// TIA Portal V17 export
// export: Created 2025-06-26T07:49:36.6585536Z, ExportSetting WithDefaults, DisplayName Totally Integrated Automation Portal, DisplayVersion V17 Update 8, DisplayName TIA Portal Openness, DisplayVersion V17 Update 8, DisplayName TIA Portal Version Control Interface, DisplayVersion V17, DisplayName STEP 7 Professional, DisplayVersion V17 Update 8, DisplayName STEP 7 Safety, DisplayVersion V17 Update 6, DisplayName WinCC Advanced, DisplayVersion V17 Update 8
FUNCTION_BLOCK "InputWarningHandling"   // FB7, FBD
TITLE = Handle I/O warnings
{ S7_Optimized_Access := 'TRUE' }
AUTHOR : Heaten
VERSION : 0.1
// stored: AutoNumber false, IsIECCheckEnabled false, IsRetainMemResEnabled false, MemoryReserve 100, SetENOAutomatically false, UDAEnableTagReadback false
   VAR
      A1101 { ExternalAccessible := 'False'; ExternalVisible := 'False'; ExternalWritable := 'False'; S7_SetPoint := 'True'} : "fbDigitalAlarm";
      A1121 { ExternalAccessible := 'False'; ExternalVisible := 'False'; ExternalWritable := 'False'; S7_SetPoint := 'True'} : "fbDigitalAlarm";
      A1140 { ExternalAccessible := 'False'; ExternalVisible := 'False'; ExternalWritable := 'False'; S7_SetPoint := 'True'} : "fbDigitalAlarm";
      A1216 { ExternalAccessible := 'False'; ExternalVisible := 'False'; ExternalWritable := 'False'; S7_SetPoint := 'True'} : "fbHMIEvent";
      A1217 { ExternalAccessible := 'False'; ExternalVisible := 'False'; ExternalWritable := 'False'; S7_SetPoint := 'True'} : "fbHMIEvent";
      A1218 { ExternalAccessible := 'False'; ExternalVisible := 'False'; ExternalWritable := 'False'; S7_SetPoint := 'True'} : "fbHMIEvent";
      A1224 { ExternalAccessible := 'False'; ExternalVisible := 'False'; ExternalWritable := 'False'; S7_SetPoint := 'True'} : "fbHMIEvent";
      A1225 { ExternalAccessible := 'False'; ExternalVisible := 'False'; ExternalWritable := 'False'; S7_SetPoint := 'True'} : "fbHMIEvent";
      A1226 { ExternalAccessible := 'False'; ExternalVisible := 'False'; ExternalWritable := 'False'; S7_SetPoint := 'True'} : "fbHMIEvent";
      A1227 { ExternalAccessible := 'False'; ExternalVisible := 'False'; ExternalWritable := 'False'; S7_SetPoint := 'True'} : "fbHMIEvent";
      A1228 { ExternalAccessible := 'False'; ExternalVisible := 'False'; ExternalWritable := 'False'; S7_SetPoint := 'True'} : "fbHMIEvent";
      A1229 { ExternalAccessible := 'False'; ExternalVisible := 'False'; ExternalWritable := 'False'; S7_SetPoint := 'True'} : "fbHMIEvent";
      A1230 { ExternalAccessible := 'False'; ExternalVisible := 'False'; ExternalWritable := 'False'; S7_SetPoint := 'True'} : "fbHMIEvent";
      A1234 { ExternalAccessible := 'False'; ExternalVisible := 'False'; ExternalWritable := 'False'; S7_SetPoint := 'True'} : "fbHMIEvent";
      A1235 { ExternalAccessible := 'False'; ExternalVisible := 'False'; ExternalWritable := 'False'; S7_SetPoint := 'True'} : "fbHMIEvent";
      A1236 { ExternalAccessible := 'False'; ExternalVisible := 'False'; ExternalWritable := 'False'; S7_SetPoint := 'True'} : "fbHMIEvent";
      A1237 { ExternalAccessible := 'False'; ExternalVisible := 'False'; ExternalWritable := 'False'; S7_SetPoint := 'True'} : "fbHMIEvent";
      A1238 { ExternalAccessible := 'False'; ExternalVisible := 'False'; ExternalWritable := 'False'; S7_SetPoint := 'True'} : "fbHMIEvent";
      A1239 { ExternalAccessible := 'False'; ExternalVisible := 'False'; ExternalWritable := 'False'; S7_SetPoint := 'True'} : "fbHMIEvent";
      A1240 { ExternalAccessible := 'False'; ExternalVisible := 'False'; ExternalWritable := 'False'; S7_SetPoint := 'True'} : "fbHMIEvent";
      A1245 { ExternalAccessible := 'False'; ExternalVisible := 'False'; ExternalWritable := 'False'; S7_SetPoint := 'True'} : "fbHMIEvent";
      A1246 { ExternalAccessible := 'False'; ExternalVisible := 'False'; ExternalWritable := 'False'; S7_SetPoint := 'True'} : "fbHMIEvent";
      A1247 { ExternalAccessible := 'False'; ExternalVisible := 'False'; ExternalWritable := 'False'; S7_SetPoint := 'True'} : "fbHMIEvent";
      A1248 { ExternalAccessible := 'False'; ExternalVisible := 'False'; ExternalWritable := 'False'; S7_SetPoint := 'True'} : "fbHMIEvent";
      A1249 { ExternalAccessible := 'False'; ExternalVisible := 'False'; ExternalWritable := 'False'; S7_SetPoint := 'True'} : "fbHMIEvent";
      A1251 { ExternalAccessible := 'False'; ExternalVisible := 'False'; ExternalWritable := 'False'; S7_SetPoint := 'True'} : "fbHMIEvent";
      A1252 { ExternalAccessible := 'False'; ExternalVisible := 'False'; ExternalWritable := 'False'; S7_SetPoint := 'True'} : "fbHMIEvent";
      A1253 { ExternalAccessible := 'False'; ExternalVisible := 'False'; ExternalWritable := 'False'; S7_SetPoint := 'True'} : "fbHMIEvent";
      A1254 { ExternalAccessible := 'False'; ExternalVisible := 'False'; ExternalWritable := 'False'; S7_SetPoint := 'True'} : "fbHMIEvent";
      A1258 { ExternalAccessible := 'False'; ExternalVisible := 'False'; ExternalWritable := 'False'; S7_SetPoint := 'True'} : "fbHMIEvent";
      A1259 { ExternalAccessible := 'False'; ExternalVisible := 'False'; ExternalWritable := 'False'; S7_SetPoint := 'True'} : "fbHMIEvent";
      A1260 { ExternalAccessible := 'False'; ExternalVisible := 'False'; ExternalWritable := 'False'; S7_SetPoint := 'True'} : "fbHMIEvent";
      A1262 { ExternalAccessible := 'False'; ExternalVisible := 'False'; ExternalWritable := 'False'; S7_SetPoint := 'True'} : "fbHMIEvent";
      A1263 { ExternalAccessible := 'False'; ExternalVisible := 'False'; ExternalWritable := 'False'; S7_SetPoint := 'True'} : "fbHMIEvent";
      A1265 { ExternalAccessible := 'False'; ExternalVisible := 'False'; ExternalWritable := 'False'; S7_SetPoint := 'True'} : "fbHMIEvent";
      A1269 { ExternalAccessible := 'False'; ExternalVisible := 'False'; ExternalWritable := 'False'; S7_SetPoint := 'True'} : "fbHMIEvent";
      A1270 { ExternalAccessible := 'False'; ExternalVisible := 'False'; ExternalWritable := 'False'; S7_SetPoint := 'True'} : "fbHMIEvent";
      A1271 { ExternalAccessible := 'False'; ExternalVisible := 'False'; ExternalWritable := 'False'; S7_SetPoint := 'True'} : "fbHMIEvent";
      A1272 { ExternalAccessible := 'False'; ExternalVisible := 'False'; ExternalWritable := 'False'; S7_SetPoint := 'True'} : "fbHMIEvent";
      A1273 { ExternalAccessible := 'False'; ExternalVisible := 'False'; ExternalWritable := 'False'; S7_SetPoint := 'True'} : "fbHMIEvent";
      A1275 { ExternalAccessible := 'False'; ExternalVisible := 'False'; ExternalWritable := 'False'; S7_SetPoint := 'True'} : "fbHMIEvent";
      A1293 { ExternalAccessible := 'False'; ExternalVisible := 'False'; ExternalWritable := 'False'; S7_SetPoint := 'True'} : "fbHMIEvent";
      A1294 { S7_SetPoint := 'True'} : "fbDigitalAlarm";
      A1295 { S7_SetPoint := 'True'} : "fbDigitalAlarm";
      A3401 { ExternalAccessible := 'False'; ExternalVisible := 'False'; ExternalWritable := 'False'; S7_SetPoint := 'True'} : "fbDigitalAlarm";
      A5200 { ExternalAccessible := 'False'; ExternalVisible := 'False'; ExternalWritable := 'False'; S7_SetPoint := 'True'} : "fbHMIEvent";
      A5201 { ExternalAccessible := 'False'; ExternalVisible := 'False'; ExternalWritable := 'False'; S7_SetPoint := 'True'} : "fbHMIEvent";
      A5202 { ExternalAccessible := 'False'; ExternalVisible := 'False'; ExternalWritable := 'False'; S7_SetPoint := 'True'} : "fbHMIEvent";
      A5203 { ExternalAccessible := 'False'; ExternalVisible := 'False'; ExternalWritable := 'False'; S7_SetPoint := 'True'} : "fbDigitalAlarm";
      A5204 { ExternalAccessible := 'False'; ExternalVisible := 'False'; ExternalWritable := 'False'; S7_SetPoint := 'True'} : "fbDigitalAlarm";
      A5206 { ExternalAccessible := 'False'; ExternalVisible := 'False'; ExternalWritable := 'False'; S7_SetPoint := 'True'} : "fbHMIEvent";
      A5256 { ExternalAccessible := 'False'; ExternalVisible := 'False'; ExternalWritable := 'False'; S7_SetPoint := 'True'} : "fbHMIEvent";
   END_VAR
BEGIN

REGION Network 1: 1101
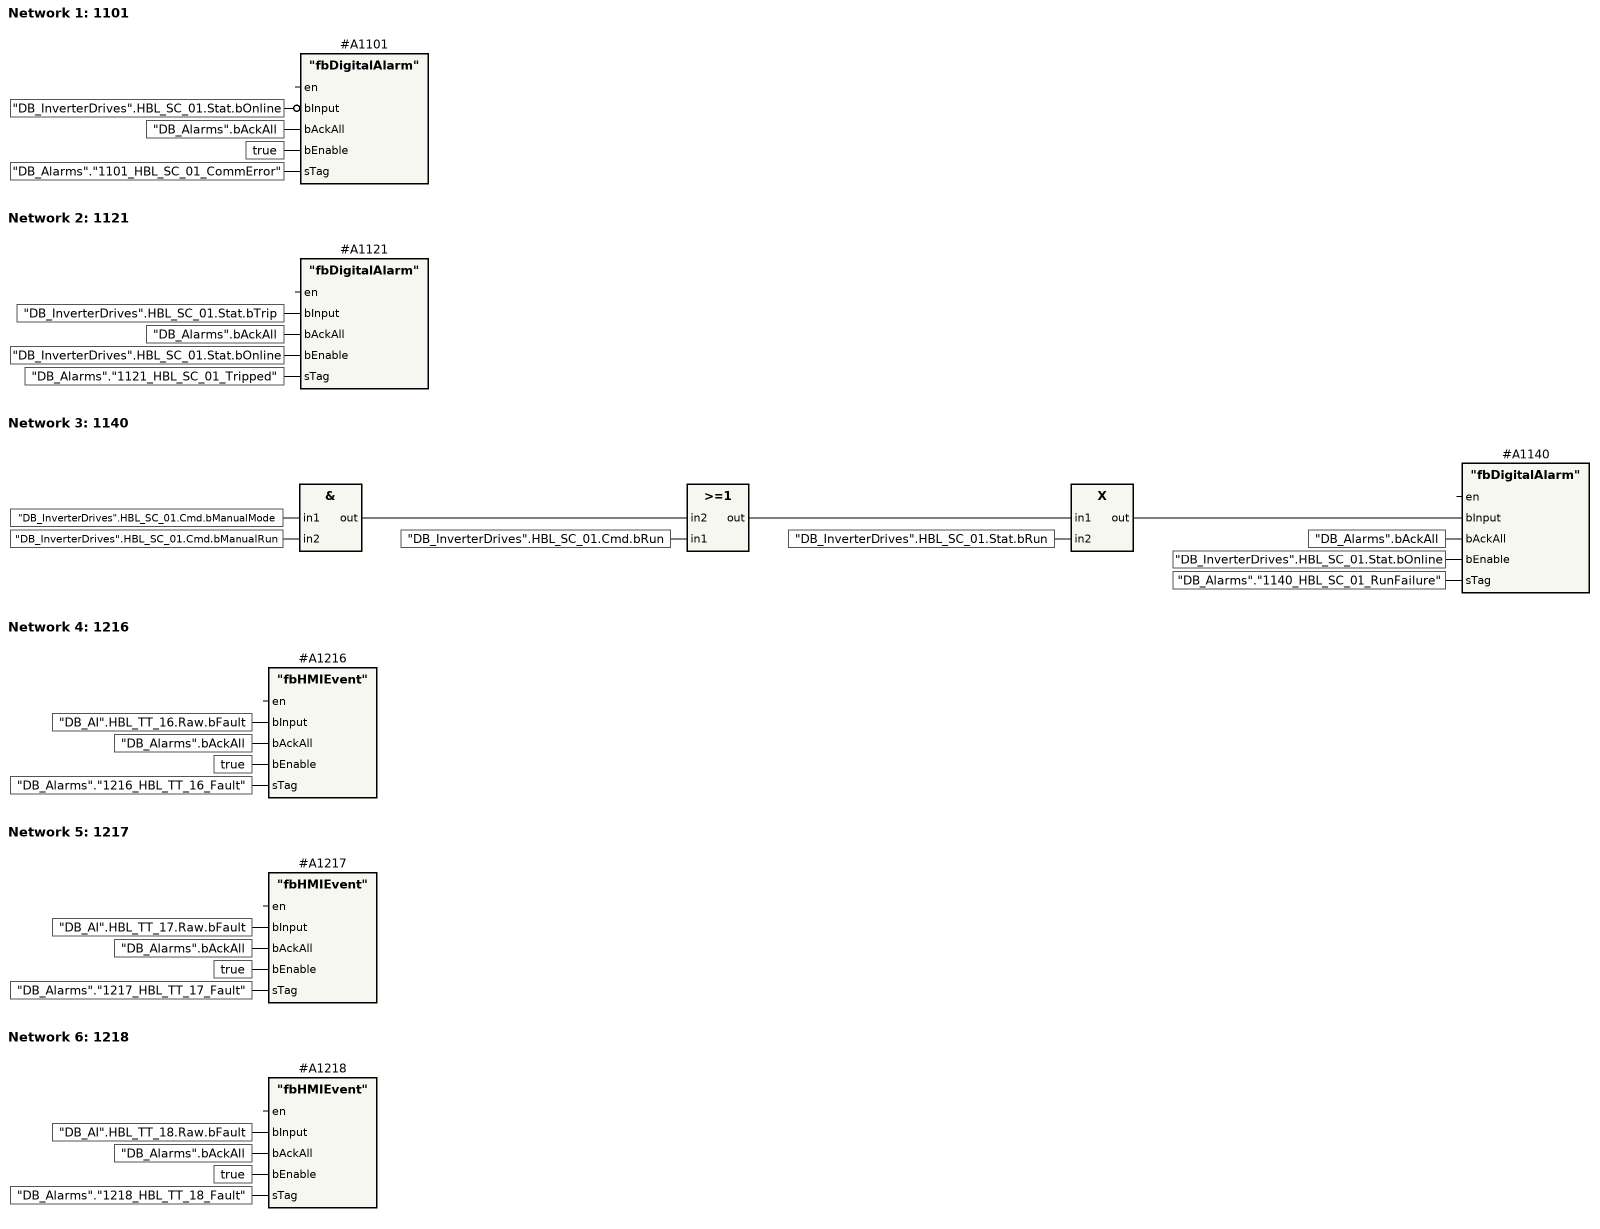
   #A1101(bInput := NOT "DB_InverterDrives".HBL_SC_01.Stat.bOnline,   // "fbDigitalAlarm"
          bAckAll := "DB_Alarms".bAckAll,
          bEnable := true,
          sTag := "DB_Alarms"."1101_HBL_SC_01_CommError");
END_REGION

REGION Network 2: 1121
   #A1121(bInput := "DB_InverterDrives".HBL_SC_01.Stat.bTrip,   // "fbDigitalAlarm"
          bAckAll := "DB_Alarms".bAckAll,
          bEnable := "DB_InverterDrives".HBL_SC_01.Stat.bOnline,
          sTag := "DB_Alarms"."1121_HBL_SC_01_Tripped");
END_REGION

REGION Network 3: 1140
   #A1140(bInput := (("DB_InverterDrives".HBL_SC_01.Cmd.bManualMode AND "DB_InverterDrives".HBL_SC_01.Cmd.bManualRun) OR "DB_InverterDrives".HBL_SC_01.Cmd.bRun) XOR "DB_InverterDrives".HBL_SC_01.Stat.bRun,   // "fbDigitalAlarm"
          bAckAll := "DB_Alarms".bAckAll,
          bEnable := "DB_InverterDrives".HBL_SC_01.Stat.bOnline,
          sTag := "DB_Alarms"."1140_HBL_SC_01_RunFailure");
END_REGION

REGION Network 4: 1216
   #A1216(bInput := "DB_AI".HBL_TT_16.Raw.bFault,   // "fbHMIEvent"
          bAckAll := "DB_Alarms".bAckAll,
          bEnable := true,
          sTag := "DB_Alarms"."1216_HBL_TT_16_Fault");
END_REGION

REGION Network 5: 1217
   #A1217(bInput := "DB_AI".HBL_TT_17.Raw.bFault,   // "fbHMIEvent"
          bAckAll := "DB_Alarms".bAckAll,
          bEnable := true,
          sTag := "DB_Alarms"."1217_HBL_TT_17_Fault");
END_REGION

REGION Network 6: 1218
   #A1218(bInput := "DB_AI".HBL_TT_18.Raw.bFault,   // "fbHMIEvent"
          bAckAll := "DB_Alarms".bAckAll,
          bEnable := true,
          sTag := "DB_Alarms"."1218_HBL_TT_18_Fault");
END_REGION

REGION Network 7: 1224
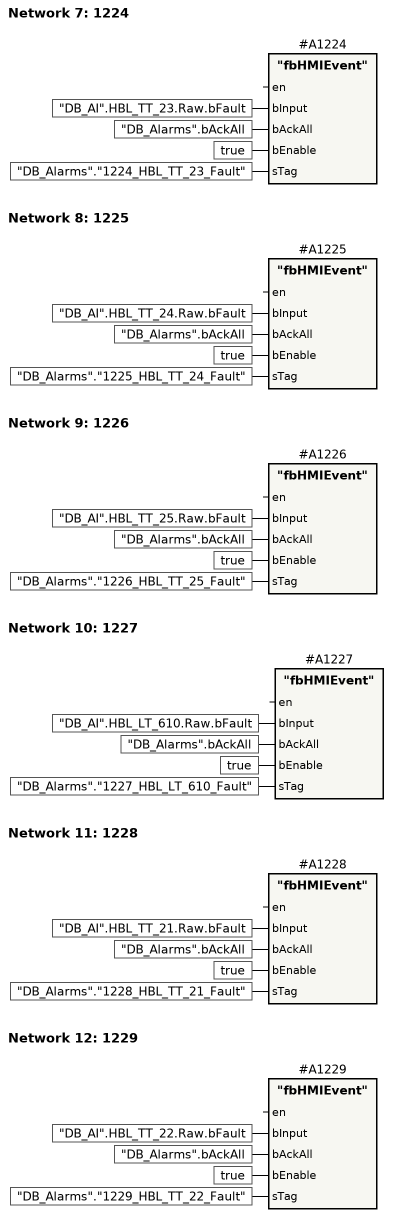
   #A1224(bInput := "DB_AI".HBL_TT_23.Raw.bFault,   // "fbHMIEvent"
          bAckAll := "DB_Alarms".bAckAll,
          bEnable := true,
          sTag := "DB_Alarms"."1224_HBL_TT_23_Fault");
END_REGION

REGION Network 8: 1225
   #A1225(bInput := "DB_AI".HBL_TT_24.Raw.bFault,   // "fbHMIEvent"
          bAckAll := "DB_Alarms".bAckAll,
          bEnable := true,
          sTag := "DB_Alarms"."1225_HBL_TT_24_Fault");
END_REGION

REGION Network 9: 1226
   #A1226(bInput := "DB_AI".HBL_TT_25.Raw.bFault,   // "fbHMIEvent"
          bAckAll := "DB_Alarms".bAckAll,
          bEnable := true,
          sTag := "DB_Alarms"."1226_HBL_TT_25_Fault");
END_REGION

REGION Network 10: 1227
   #A1227(bInput := "DB_AI".HBL_LT_610.Raw.bFault,   // "fbHMIEvent"
          bAckAll := "DB_Alarms".bAckAll,
          bEnable := true,
          sTag := "DB_Alarms"."1227_HBL_LT_610_Fault");
END_REGION

REGION Network 11: 1228
   #A1228(bInput := "DB_AI".HBL_TT_21.Raw.bFault,   // "fbHMIEvent"
          bAckAll := "DB_Alarms".bAckAll,
          bEnable := true,
          sTag := "DB_Alarms"."1228_HBL_TT_21_Fault");
END_REGION

REGION Network 12: 1229
   #A1229(bInput := "DB_AI".HBL_TT_22.Raw.bFault,   // "fbHMIEvent"
          bAckAll := "DB_Alarms".bAckAll,
          bEnable := true,
          sTag := "DB_Alarms"."1229_HBL_TT_22_Fault");
END_REGION

REGION Network 13: 1230
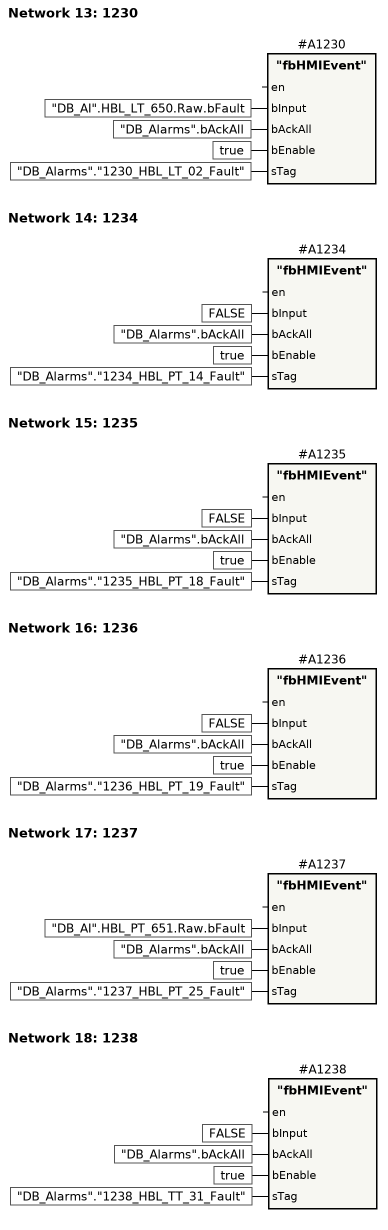
   #A1230(bInput := "DB_AI".HBL_LT_650.Raw.bFault,   // "fbHMIEvent"
          bAckAll := "DB_Alarms".bAckAll,
          bEnable := true,
          sTag := "DB_Alarms"."1230_HBL_LT_02_Fault");
END_REGION

REGION Network 14: 1234
   #A1234(bInput := FALSE,   // "fbHMIEvent"
          bAckAll := "DB_Alarms".bAckAll,
          bEnable := true,
          sTag := "DB_Alarms"."1234_HBL_PT_14_Fault");
END_REGION

REGION Network 15: 1235
   #A1235(bInput := FALSE,   // "fbHMIEvent"
          bAckAll := "DB_Alarms".bAckAll,
          bEnable := true,
          sTag := "DB_Alarms"."1235_HBL_PT_18_Fault");
END_REGION

REGION Network 16: 1236
   #A1236(bInput := FALSE,   // "fbHMIEvent"
          bAckAll := "DB_Alarms".bAckAll,
          bEnable := true,
          sTag := "DB_Alarms"."1236_HBL_PT_19_Fault");
END_REGION

REGION Network 17: 1237
   #A1237(bInput := "DB_AI".HBL_PT_651.Raw.bFault,   // "fbHMIEvent"
          bAckAll := "DB_Alarms".bAckAll,
          bEnable := true,
          sTag := "DB_Alarms"."1237_HBL_PT_25_Fault");
END_REGION

REGION Network 18: 1238
   #A1238(bInput := FALSE,   // "fbHMIEvent"
          bAckAll := "DB_Alarms".bAckAll,
          bEnable := true,
          sTag := "DB_Alarms"."1238_HBL_TT_31_Fault");
END_REGION

REGION Network 19: 1239
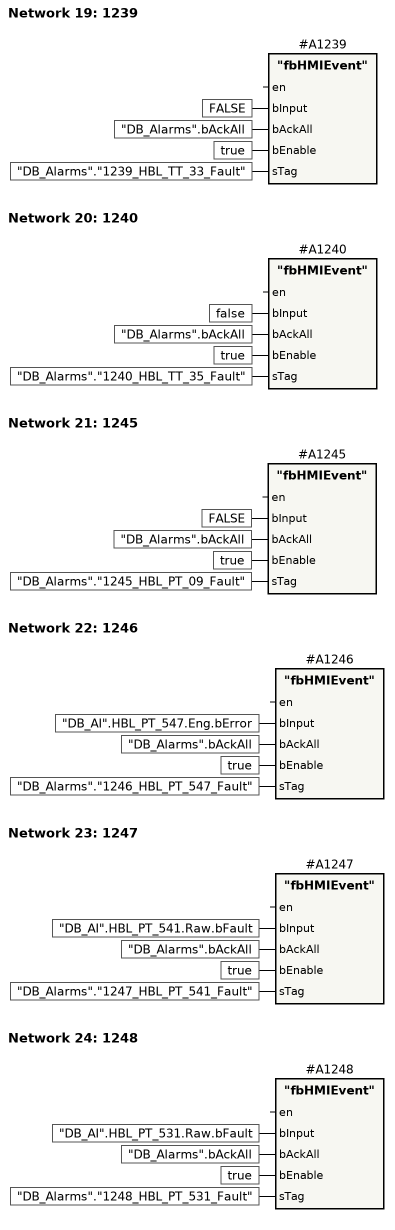
   #A1239(bInput := FALSE,   // "fbHMIEvent"
          bAckAll := "DB_Alarms".bAckAll,
          bEnable := true,
          sTag := "DB_Alarms"."1239_HBL_TT_33_Fault");
END_REGION

REGION Network 20: 1240
   #A1240(bInput := false,   // "fbHMIEvent"
          bAckAll := "DB_Alarms".bAckAll,
          bEnable := true,
          sTag := "DB_Alarms"."1240_HBL_TT_35_Fault");
END_REGION

REGION Network 21: 1245
   #A1245(bInput := FALSE,   // "fbHMIEvent"
          bAckAll := "DB_Alarms".bAckAll,
          bEnable := true,
          sTag := "DB_Alarms"."1245_HBL_PT_09_Fault");
END_REGION

REGION Network 22: 1246
   #A1246(bInput := "DB_AI".HBL_PT_547.Eng.bError,   // "fbHMIEvent"
          bAckAll := "DB_Alarms".bAckAll,
          bEnable := true,
          sTag := "DB_Alarms"."1246_HBL_PT_547_Fault");
END_REGION

REGION Network 23: 1247
   #A1247(bInput := "DB_AI".HBL_PT_541.Raw.bFault,   // "fbHMIEvent"
          bAckAll := "DB_Alarms".bAckAll,
          bEnable := true,
          sTag := "DB_Alarms"."1247_HBL_PT_541_Fault");
END_REGION

REGION Network 24: 1248
   #A1248(bInput := "DB_AI".HBL_PT_531.Raw.bFault,   // "fbHMIEvent"
          bAckAll := "DB_Alarms".bAckAll,
          bEnable := true,
          sTag := "DB_Alarms"."1248_HBL_PT_531_Fault");
END_REGION

REGION Network 25: 1249
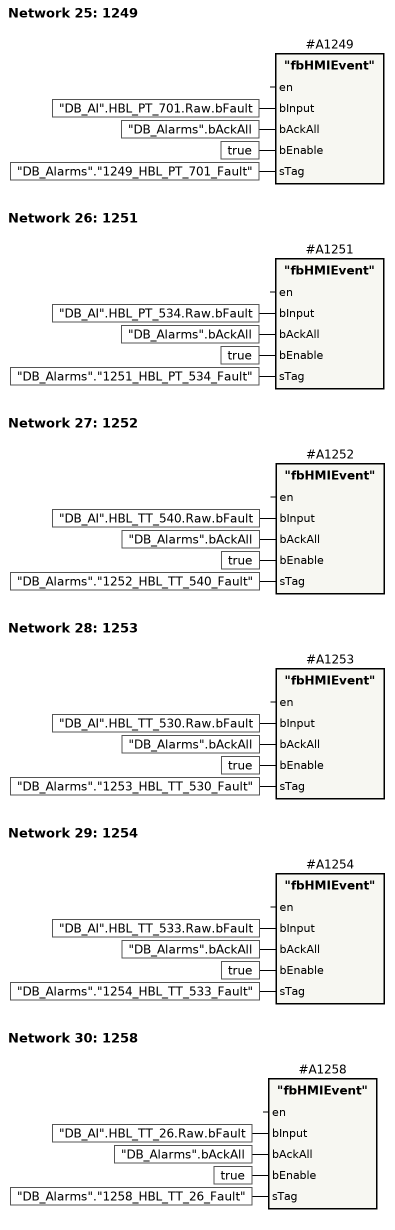
   #A1249(bInput := "DB_AI".HBL_PT_701.Raw.bFault,   // "fbHMIEvent"
          bAckAll := "DB_Alarms".bAckAll,
          bEnable := true,
          sTag := "DB_Alarms"."1249_HBL_PT_701_Fault");
END_REGION

REGION Network 26: 1251
   #A1251(bInput := "DB_AI".HBL_PT_534.Raw.bFault,   // "fbHMIEvent"
          bAckAll := "DB_Alarms".bAckAll,
          bEnable := true,
          sTag := "DB_Alarms"."1251_HBL_PT_534_Fault");
END_REGION

REGION Network 27: 1252
   #A1252(bInput := "DB_AI".HBL_TT_540.Raw.bFault,   // "fbHMIEvent"
          bAckAll := "DB_Alarms".bAckAll,
          bEnable := true,
          sTag := "DB_Alarms"."1252_HBL_TT_540_Fault");
END_REGION

REGION Network 28: 1253
   #A1253(bInput := "DB_AI".HBL_TT_530.Raw.bFault,   // "fbHMIEvent"
          bAckAll := "DB_Alarms".bAckAll,
          bEnable := true,
          sTag := "DB_Alarms"."1253_HBL_TT_530_Fault");
END_REGION

REGION Network 29: 1254
   #A1254(bInput := "DB_AI".HBL_TT_533.Raw.bFault,   // "fbHMIEvent"
          bAckAll := "DB_Alarms".bAckAll,
          bEnable := true,
          sTag := "DB_Alarms"."1254_HBL_TT_533_Fault");
END_REGION

REGION Network 30: 1258
   #A1258(bInput := "DB_AI".HBL_TT_26.Raw.bFault,   // "fbHMIEvent"
          bAckAll := "DB_Alarms".bAckAll,
          bEnable := true,
          sTag := "DB_Alarms"."1258_HBL_TT_26_Fault");
END_REGION

REGION Network 31: 1259
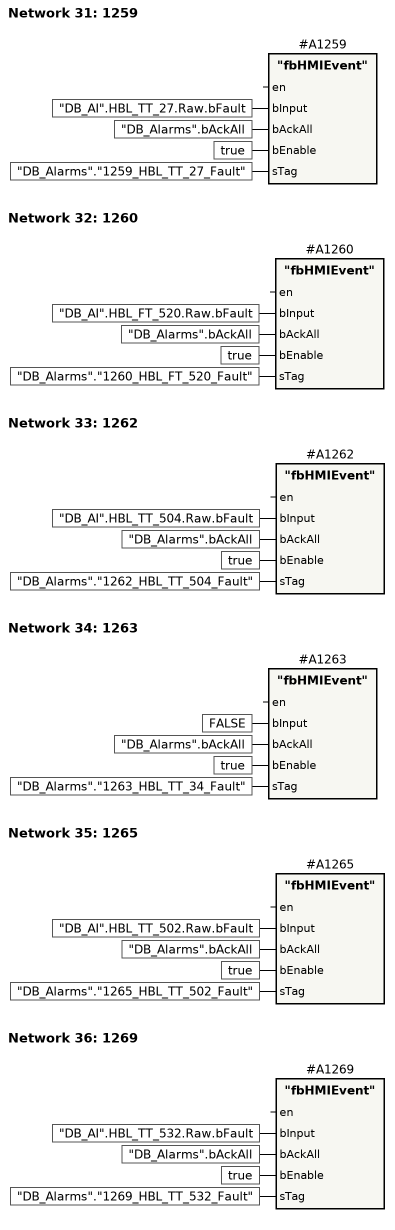
   #A1259(bInput := "DB_AI".HBL_TT_27.Raw.bFault,   // "fbHMIEvent"
          bAckAll := "DB_Alarms".bAckAll,
          bEnable := true,
          sTag := "DB_Alarms"."1259_HBL_TT_27_Fault");
END_REGION

REGION Network 32: 1260
   #A1260(bInput := "DB_AI".HBL_FT_520.Raw.bFault,   // "fbHMIEvent"
          bAckAll := "DB_Alarms".bAckAll,
          bEnable := true,
          sTag := "DB_Alarms"."1260_HBL_FT_520_Fault");
END_REGION

REGION Network 33: 1262
   #A1262(bInput := "DB_AI".HBL_TT_504.Raw.bFault,   // "fbHMIEvent"
          bAckAll := "DB_Alarms".bAckAll,
          bEnable := true,
          sTag := "DB_Alarms"."1262_HBL_TT_504_Fault");
END_REGION

REGION Network 34: 1263
   #A1263(bInput := FALSE,   // "fbHMIEvent"
          bAckAll := "DB_Alarms".bAckAll,
          bEnable := true,
          sTag := "DB_Alarms"."1263_HBL_TT_34_Fault");
END_REGION

REGION Network 35: 1265
   #A1265(bInput := "DB_AI".HBL_TT_502.Raw.bFault,   // "fbHMIEvent"
          bAckAll := "DB_Alarms".bAckAll,
          bEnable := true,
          sTag := "DB_Alarms"."1265_HBL_TT_502_Fault");
END_REGION

REGION Network 36: 1269
   #A1269(bInput := "DB_AI".HBL_TT_532.Raw.bFault,   // "fbHMIEvent"
          bAckAll := "DB_Alarms".bAckAll,
          bEnable := true,
          sTag := "DB_Alarms"."1269_HBL_TT_532_Fault");
END_REGION

REGION Network 37: 1270
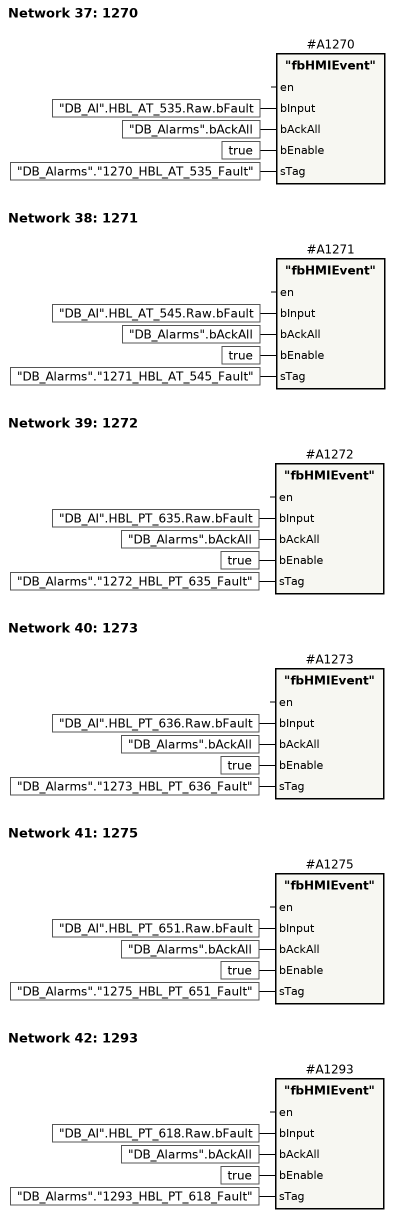
   #A1270(bInput := "DB_AI".HBL_AT_535.Raw.bFault,   // "fbHMIEvent"
          bAckAll := "DB_Alarms".bAckAll,
          bEnable := true,
          sTag := "DB_Alarms"."1270_HBL_AT_535_Fault");
END_REGION

REGION Network 38: 1271
   #A1271(bInput := "DB_AI".HBL_AT_545.Raw.bFault,   // "fbHMIEvent"
          bAckAll := "DB_Alarms".bAckAll,
          bEnable := true,
          sTag := "DB_Alarms"."1271_HBL_AT_545_Fault");
END_REGION

REGION Network 39: 1272
   #A1272(bInput := "DB_AI".HBL_PT_635.Raw.bFault,   // "fbHMIEvent"
          bAckAll := "DB_Alarms".bAckAll,
          bEnable := true,
          sTag := "DB_Alarms"."1272_HBL_PT_635_Fault");
END_REGION

REGION Network 40: 1273
   #A1273(bInput := "DB_AI".HBL_PT_636.Raw.bFault,   // "fbHMIEvent"
          bAckAll := "DB_Alarms".bAckAll,
          bEnable := true,
          sTag := "DB_Alarms"."1273_HBL_PT_636_Fault");
END_REGION

REGION Network 41: 1275
   #A1275(bInput := "DB_AI".HBL_PT_651.Raw.bFault,   // "fbHMIEvent"
          bAckAll := "DB_Alarms".bAckAll,
          bEnable := true,
          sTag := "DB_Alarms"."1275_HBL_PT_651_Fault");
END_REGION

REGION Network 42: 1293
   #A1293(bInput := "DB_AI".HBL_PT_618.Raw.bFault,   // "fbHMIEvent"
          bAckAll := "DB_Alarms".bAckAll,
          bEnable := true,
          sTag := "DB_Alarms"."1293_HBL_PT_618_Fault");
END_REGION

REGION Network 43: 1294
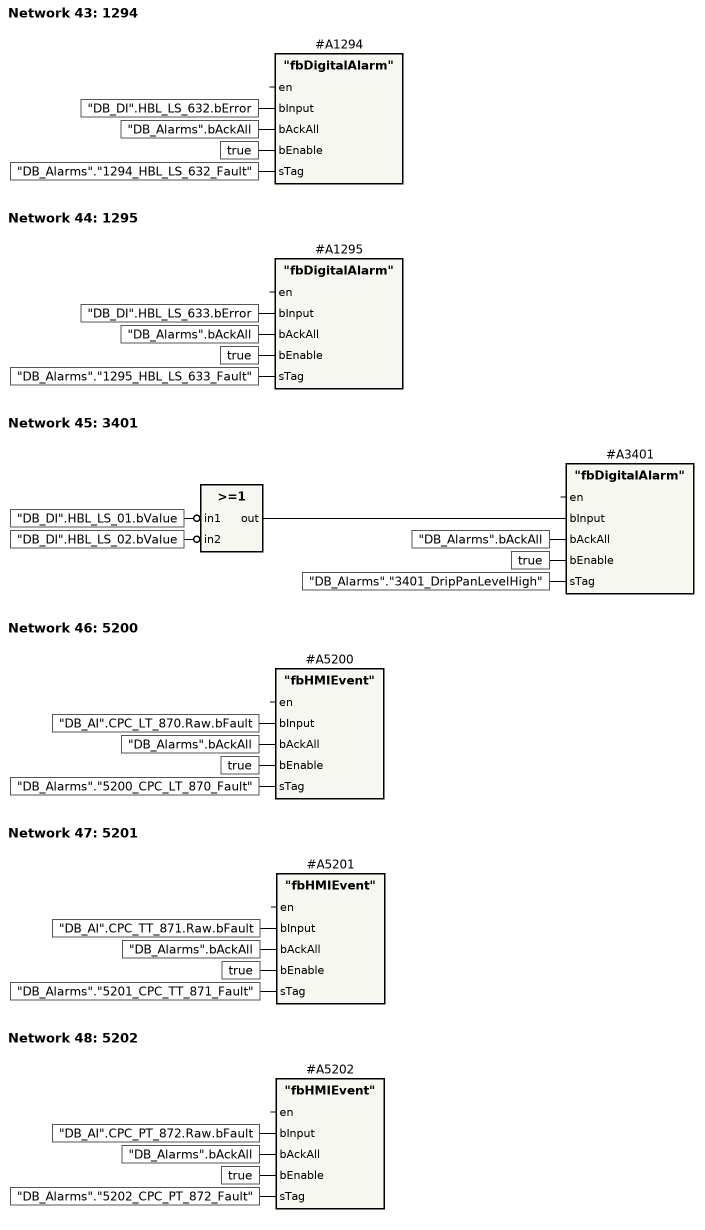
   #A1294(bInput := "DB_DI".HBL_LS_632.bError,   // "fbDigitalAlarm"
          bAckAll := "DB_Alarms".bAckAll,
          bEnable := true,
          sTag := "DB_Alarms"."1294_HBL_LS_632_Fault");
END_REGION

REGION Network 44: 1295
   #A1295(bInput := "DB_DI".HBL_LS_633.bError,   // "fbDigitalAlarm"
          bAckAll := "DB_Alarms".bAckAll,
          bEnable := true,
          sTag := "DB_Alarms"."1295_HBL_LS_633_Fault");
END_REGION

REGION Network 45: 3401
   #A3401(bInput := NOT "DB_DI".HBL_LS_01.bValue OR NOT "DB_DI".HBL_LS_02.bValue,   // "fbDigitalAlarm"
          bAckAll := "DB_Alarms".bAckAll,
          bEnable := true,
          sTag := "DB_Alarms"."3401_DripPanLevelHigh");
END_REGION

REGION Network 46: 5200
   #A5200(bInput := "DB_AI".CPC_LT_870.Raw.bFault,   // "fbHMIEvent"
          bAckAll := "DB_Alarms".bAckAll,
          bEnable := true,
          sTag := "DB_Alarms"."5200_CPC_LT_870_Fault");
END_REGION

REGION Network 47: 5201
   #A5201(bInput := "DB_AI".CPC_TT_871.Raw.bFault,   // "fbHMIEvent"
          bAckAll := "DB_Alarms".bAckAll,
          bEnable := true,
          sTag := "DB_Alarms"."5201_CPC_TT_871_Fault");
END_REGION

REGION Network 48: 5202
   #A5202(bInput := "DB_AI".CPC_PT_872.Raw.bFault,   // "fbHMIEvent"
          bAckAll := "DB_Alarms".bAckAll,
          bEnable := true,
          sTag := "DB_Alarms"."5202_CPC_PT_872_Fault");
END_REGION

REGION Network 49: 5203
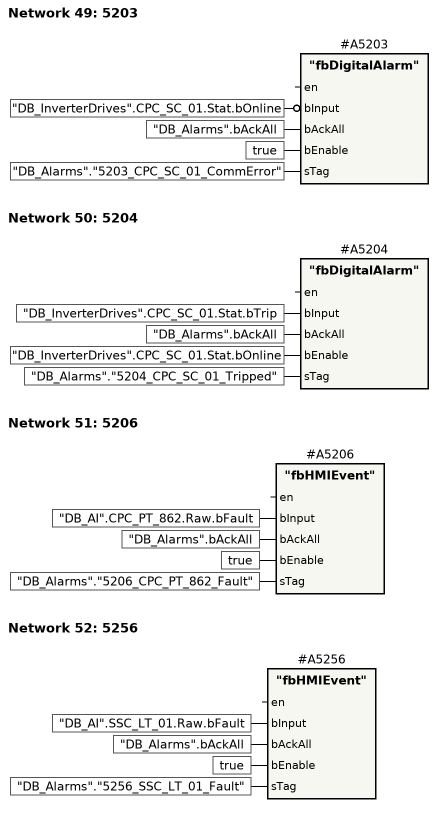
   #A5203(bInput := NOT "DB_InverterDrives".CPC_SC_01.Stat.bOnline,   // "fbDigitalAlarm"
          bAckAll := "DB_Alarms".bAckAll,
          bEnable := true,
          sTag := "DB_Alarms"."5203_CPC_SC_01_CommError");
END_REGION

REGION Network 50: 5204
   // Only show if online
   #A5204(bInput := "DB_InverterDrives".CPC_SC_01.Stat.bTrip,   // "fbDigitalAlarm"
          bAckAll := "DB_Alarms".bAckAll,
          bEnable := "DB_InverterDrives".CPC_SC_01.Stat.bOnline,
          sTag := "DB_Alarms"."5204_CPC_SC_01_Tripped");
END_REGION

REGION Network 51: 5206
   #A5206(bInput := "DB_AI".CPC_PT_862.Raw.bFault,   // "fbHMIEvent"
          bAckAll := "DB_Alarms".bAckAll,
          bEnable := true,
          sTag := "DB_Alarms"."5206_CPC_PT_862_Fault");
END_REGION

REGION Network 52: 5256
   #A5256(bInput := "DB_AI".SSC_LT_01.Raw.bFault,   // "fbHMIEvent"
          bAckAll := "DB_Alarms".bAckAll,
          bEnable := true,
          sTag := "DB_Alarms"."5256_SSC_LT_01_Fault");
END_REGION
END_FUNCTION_BLOCK
